// Mitsubishi GX Works2 project: TH15   PLC: FX2N/FX2NC

PROGRAM MAIN
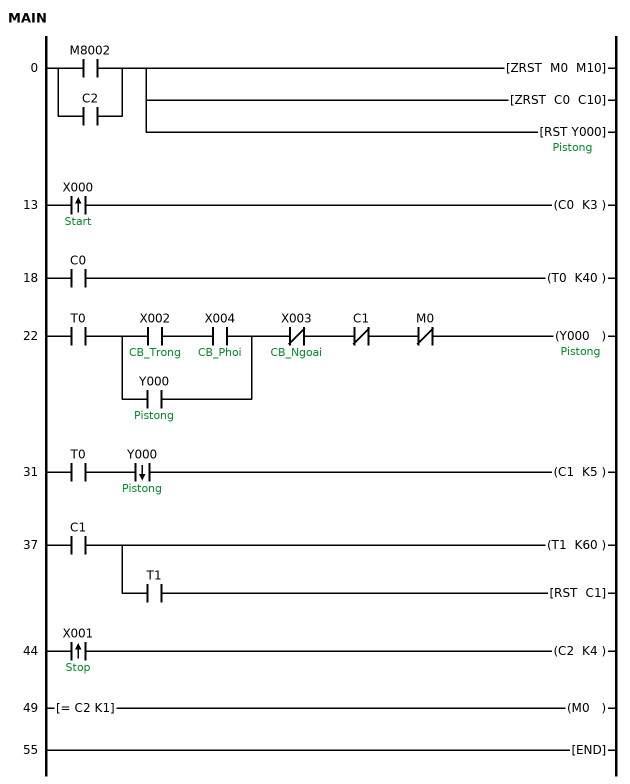
0     LD      M8002
      OR      C2
      ZRST    M0 M10
      ZRST    C0 C10
      RST     Y000  ; Pistong
13    LDP     X000  ; Start
      OUT     C0 K3
18    LD      C0
      OUT     T0 K40
22    LD      T0
      LD      X002  ; CB_Trong
      AND     X004  ; CB_Phoi
      OR      Y000  ; Pistong
      ANB
      ANI     X003  ; CB_Ngoai
      ANI     C1
      ANI     M0
      OUT     Y000  ; Pistong
31    LD      T0
      ANDF    Y000  ; Pistong
      OUT     C1 K5
37    LD      C1
      OUT     T1 K60
      AND     T1
      RST     C1
44    LDP     X001  ; Stop
      OUT     C2 K4
49    LD=     C2 K1
      OUT     M0
55    END
END_PROGRAM
